FUNCTION_BLOCK SM_LinearAxis EXTENDS BaseAxis
VAR_INPUT
END_VAR
VAR_OUTPUT
	///Actual position of the axis
	{attribute 'OPC.UA.DA' := '1'}
	{attribute 'OPC.UA.DA.Access' := '1'}
	actPos: LinearPosition;
	///Actual velocity of the axis
	{attribute 'OPC.UA.DA' := '1'}
	{attribute 'OPC.UA.DA.Access' := '1'}
	actVel: LinearVelocity;
END_VAR
VAR_IN_OUT
END_VAR
VAR
END_VAR

actPos( newMillimetersValue := axis_ref.NcToPlc.ActPos );
actVel( newMillimetersPerSecondValue := axis_ref.NcToPlc.ActVelo );
SUPER^();

END_FUNCTION_BLOCK

(* stored: Version 1.1.0.1, ProductVersion 3.1.4019.2
   POU SM_LinearAxis: Id {c82c0b0a-65a5-4aca-bc76-f4445f6a15ce}, SpecialFunc None *)
